FUNCTION F_WRITE_MEMORY : BOOL
VAR_INPUT
	cbData : UDINT;
	pData : POINTER TO BYTE;
	cbBuffer : UDINT;
	pBuffer : POINTER TO BYTE;
END_VAR
VAR
END_VAR

FW_MemMove(pDest:=pBuffer + cbData,pSrc:=pBuffer,cbLen:=cbBuffer-cbData);

FW_MemMove(pDest:=pBuffer,pSrc:=pData,cbLen:=cbData);

END_FUNCTION

(* stored: Version 1.1.0.1, ProductVersion 3.1.4022.12
   POU F_WRITE_MEMORY: Id {9508e750-2377-4d61-b7ae-cade5d933b3d}, SpecialFunc None *)
